{attribute addProperty BoxType "EP6601-0002-0018"}
{attribute addProperty Id "InfoDataInfoData_BC63D37F8010"}
{attribute addProperty CRC "424293389"}
{attribute addProperty SizeInBites "80"}
{attribute addProperty SizeInBytes "10"}
TYPE EP6601_194A340D :
STRUCT
	{attribute addProperty Name "InfoData"}
	InfoData : InfoData_BC63D37F;
END_STRUCT
END_TYPE

(* stored: Version 1.2.0.0, ProductVersion 3.1.4024.9
   DUT EP6601_194A340D: Id {963699f9-44d4-46e2-93f7-3c9dcdee578f} *)
